// TIA Portal V16 export
// export: Created 2021-11-12T13:32:30.1971542Z, ExportSetting WithDefaults, DisplayName Totally Integrated Automation Portal, DisplayVersion V16 Update 3, DisplayName TIA Portal Version Control Interface, DisplayVersion V16 Update 2, DisplayName TIA Portal Openness, DisplayVersion V16 Update 3, DisplayName SINAMICS Startdrive Advanced, DisplayVersion V16 Update 5, DisplayName SINAMICS Startdrive G130, G150, S120, S150, SINAMICS MV, S210, DisplayVersion V16 Update 5, DisplayName SINAMICS Startdrive G110M, G120, G120C, G120D, G120P, G115D, DisplayVersion V16 Update 5, DisplayName STEP 7 Professional, DisplayVersion V16 Update 3, DisplayName STEP 7 Safety, DisplayVersion V16, DisplayName WinCC UA Professional, DisplayVersion V16 Update 3
DATA_BLOCK "IDB_Station1R3"   // DB164
VERSION : 0.1
// stored: AutoNumber true, DBAccessibleFromOPCUA true, InstanceOfName Station1R3, InstanceOfType FB
"Station1R3"
   // VAR
   //    SF_RO01_Timeout : "STD_DI_Mon";
   //    SF_RO01_Lubrication : "STD_DI_Mon";
   //    SF_RC01 : "STD_DriveRobotABB";
   //    SF_RO01 : "STD_RobotABB";
   //    SF_RobotGripper : "STD_RobotGripper";
   //    SF_Sequence { S7_SetPoint := 'True'} : "Station 1R3 Seq";
   //    SF_Lubrication { S7_SetPoint := 'True'} : "TrackLubrication";
   //    SF_RobNotUsed { S7_SetPoint := 'True'} : "STD_OnOff";
   //    SS_RobotZones { S7_SetPoint := 'True'} : "STD_RobotZones";
   //    SS_Edge { S7_SetPoint := 'True'} : Array[0..100] of Bool;
   //    SDIPartId : DInt;
   //    SI_PartType : Int;
   //    SI_130RowNo { ExternalAccessible := 'False'; ExternalVisible := 'False'; ExternalWritable := 'False'} : Int;
   //    SI_130LineNo { ExternalAccessible := 'False'; ExternalVisible := 'False'; ExternalWritable := 'False'} : Int;
   //    SI_150RowNo { ExternalAccessible := 'False'; ExternalVisible := 'False'; ExternalWritable := 'False'} : Int;
   //    SI_150LineNo { ExternalAccessible := 'False'; ExternalVisible := 'False'; ExternalWritable := 'False'} : Int;
   //    SI_170RowNo { ExternalAccessible := 'False'; ExternalVisible := 'False'; ExternalWritable := 'False'} : Int;
   //    SI_170LineNo { ExternalAccessible := 'False'; ExternalVisible := 'False'; ExternalWritable := 'False'} : Int;
   //    SB1TakePosFound130 { ExternalAccessible := 'False'; ExternalVisible := 'False'; ExternalWritable := 'False'} : Bool;
   //    SB1PutPosFound150 { ExternalAccessible := 'False'; ExternalVisible := 'False'; ExternalWritable := 'False'} : Bool;
   //    SB1PutPosFound170 { ExternalAccessible := 'False'; ExternalVisible := 'False'; ExternalWritable := 'False'} : Bool;
   //    SB1ReqToChangeTool : Bool;
   //    SB1ChangeToolDone : Bool;
   //    SB1CycleAutostop : Bool;
   //    SB1ServicePosReq { ExternalAccessible := 'False'; ExternalVisible := 'False'; ExternalWritable := 'False'} : Bool;
   //    SB1LubricError : Bool;
   //    SB1Robot1Initialized : Bool;
   //    SB1Robot2Initialized : Bool;
   // END_VAR
BEGIN
END_DATA_BLOCK
